// Mitsubishi GX Works2 project: 등가회로   PLC: Q02/Q02H

PROGRAM MAIN
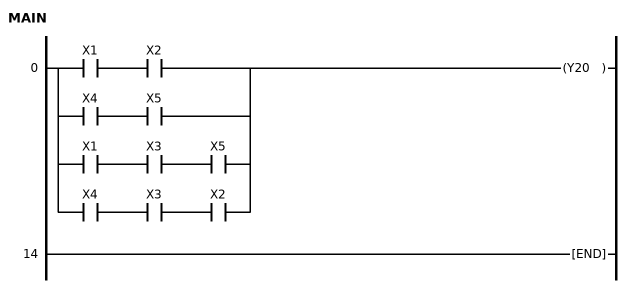
0     LD      X1
      AND     X2
      LD      X4
      AND     X5
      ORB
      LD      X1
      AND     X3
      AND     X5
      ORB
      LD      X4
      AND     X3
      AND     X2
      ORB
      OUT     Y20
14    END
END_PROGRAM
